% RSLogix 500 project Mixing_Room_1980_Kettle_original_backup_Aug_20_2021.RSS, saved by version 11.00.00.00 %
PROJECT "UNTITLED"    % processor: MicroLogix 1200 %

PROGRAM FILES
  LAD 2   55 rungs

DATA FILES
  O0 OUTPUT  8 elements
  I1 INPUT  13 elements
  S2 STATUS  66 elements
  B3 BINARY  5 elements
  T4 TIMER  5 elements
  C5 COUNTER  1 elements
  R6 CONTROL  1 elements
  N7 INTEGER  60 elements
  F8 FLOAT  141 elements
  PD9   1 elements

LADDER 2
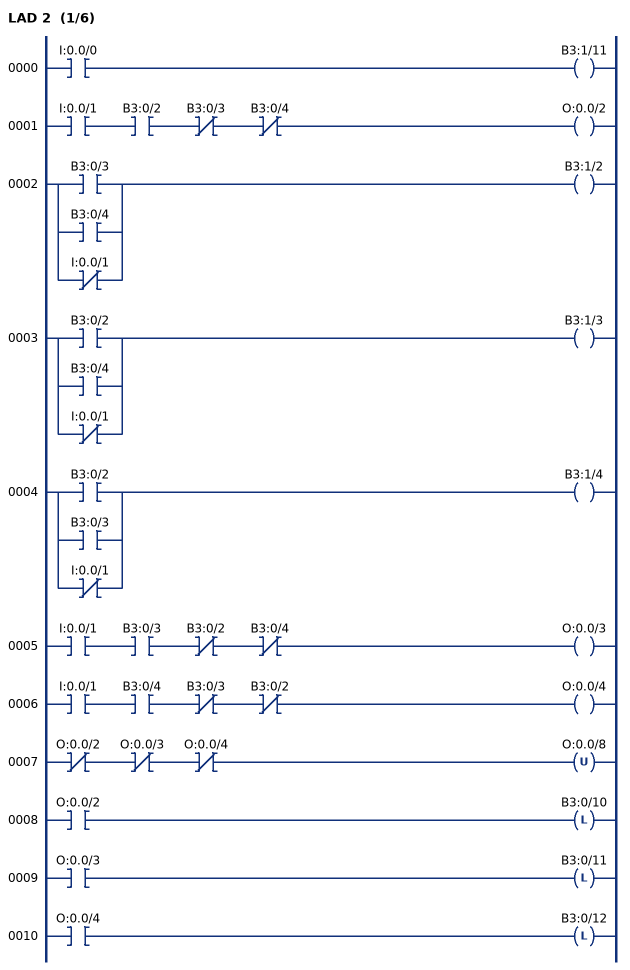
% Rung: 0 %
SOR XIC I:0.0/0 OTE B3:1/11 EOR
% Rung: 1 %
SOR XIC I:0.0/1 XIC B3:0/2 XIO B3:0/3 XIO B3:0/4 OTE O:0.0/2 EOR
% Rung: 2 %
SOR BST XIC B3:0/3 NXB BST XIC B3:0/4 NXB XIO I:0.0/1 BND BND OTE B3:1/2 EOR
% Rung: 3 %
SOR BST XIC B3:0/2 NXB BST XIC B3:0/4 NXB XIO I:0.0/1 BND BND OTE B3:1/3 EOR
% Rung: 4 %
SOR BST XIC B3:0/2 NXB BST XIC B3:0/3 NXB XIO I:0.0/1 BND BND OTE B3:1/4 EOR
% Rung: 5 %
SOR XIC I:0.0/1 XIC B3:0/3 XIO B3:0/2 XIO B3:0/4 OTE O:0.0/3 EOR
% Rung: 6 %
SOR XIC I:0.0/1 XIC B3:0/4 XIO B3:0/3 XIO B3:0/2 OTE O:0.0/4 EOR
% Rung: 7 %
SOR XIO O:0.0/2 XIO O:0.0/3 XIO O:0.0/4 OTU O:0.0/8 EOR
% Rung: 8 %
SOR XIC O:0.0/2 OTL B3:0/10 EOR
% Rung: 9 %
SOR XIC O:0.0/3 OTL B3:0/11 EOR
% Rung: 10 %
SOR XIC O:0.0/4 OTL B3:0/12 EOR

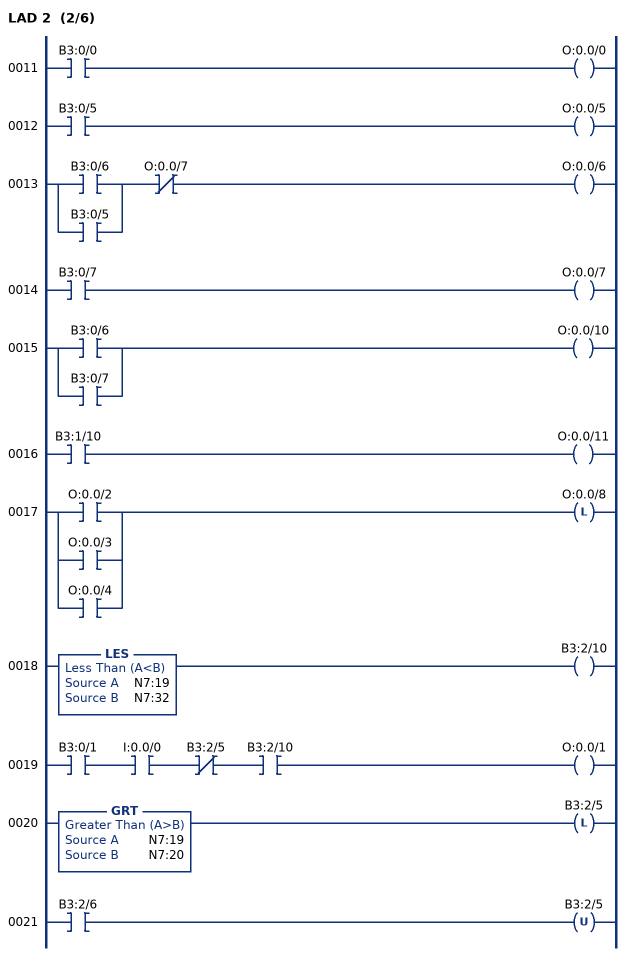
% Rung: 11 %
SOR XIC B3:0/0 OTE O:0.0/0 EOR
% Rung: 12 %
SOR XIC B3:0/5 OTE O:0.0/5 EOR
% Rung: 13 %
SOR BST XIC B3:0/6 NXB XIC B3:0/5 BND XIO O:0.0/7 OTE O:0.0/6 EOR
% Rung: 14 %
SOR XIC B3:0/7 OTE O:0.0/7 EOR
% Rung: 15 %
SOR BST XIC B3:0/6 NXB XIC B3:0/7 BND OTE O:0.0/10 EOR
% Rung: 16 %
SOR XIC B3:1/10 OTE O:0.0/11 EOR
% Rung: 17 %
SOR BST XIC O:0.0/2 NXB BST XIC O:0.0/3 NXB XIC O:0.0/4 BND BND OTL O:0.0/8 EOR
% Rung: 18 %
SOR LES N7:19 N7:32 OTE B3:2/10 EOR
% Rung: 19 %
SOR XIC B3:0/1 XIC I:0.0/0 XIO B3:2/5 XIC B3:2/10 OTE O:0.0/1 EOR
% Rung: 20 %
SOR GRT N7:19 N7:20 OTL B3:2/5 EOR
% Rung: 21 %
SOR XIC B3:2/6 OTU B3:2/5 EOR

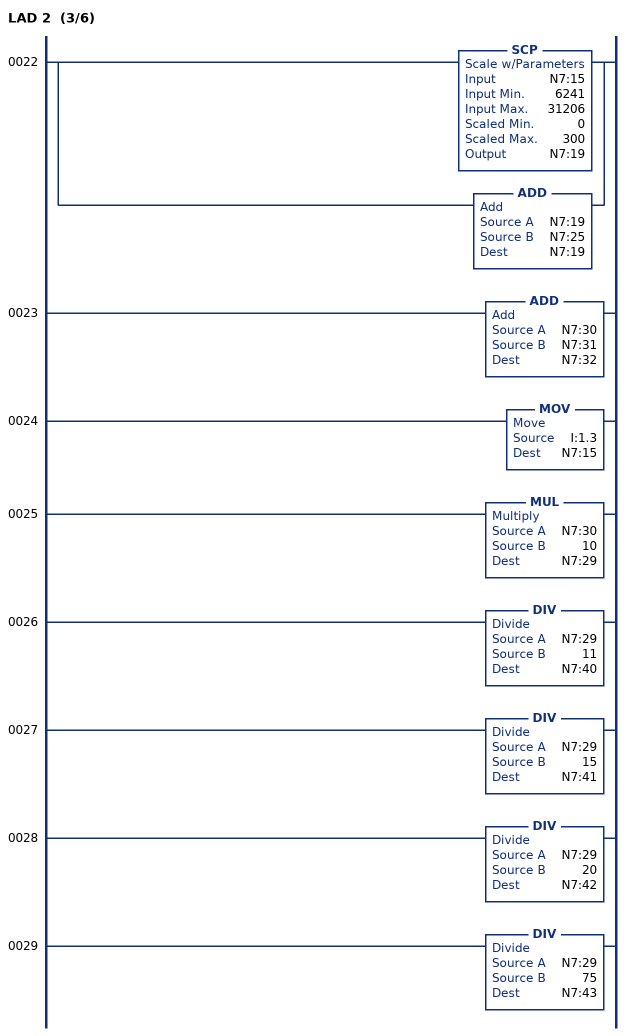
% Rung: 22 %
SOR BST SCP N7:15 6241 31206 0 300 N7:19 NXB ADD N7:19 N7:25 N7:19 BND EOR
% Rung: 23 %
SOR ADD N7:30 N7:31 N7:32 EOR
% Rung: 24 %
SOR MOV I:1.3 N7:15 EOR
% Rung: 25 %
SOR MUL N7:30 10 N7:29 EOR
% Rung: 26 %
SOR DIV N7:29 11 N7:40 EOR
% Rung: 27 %
SOR DIV N7:29 15 N7:41 EOR
% Rung: 28 %
SOR DIV N7:29 20 N7:42 EOR
% Rung: 29 %
SOR DIV N7:29 75 N7:43 EOR

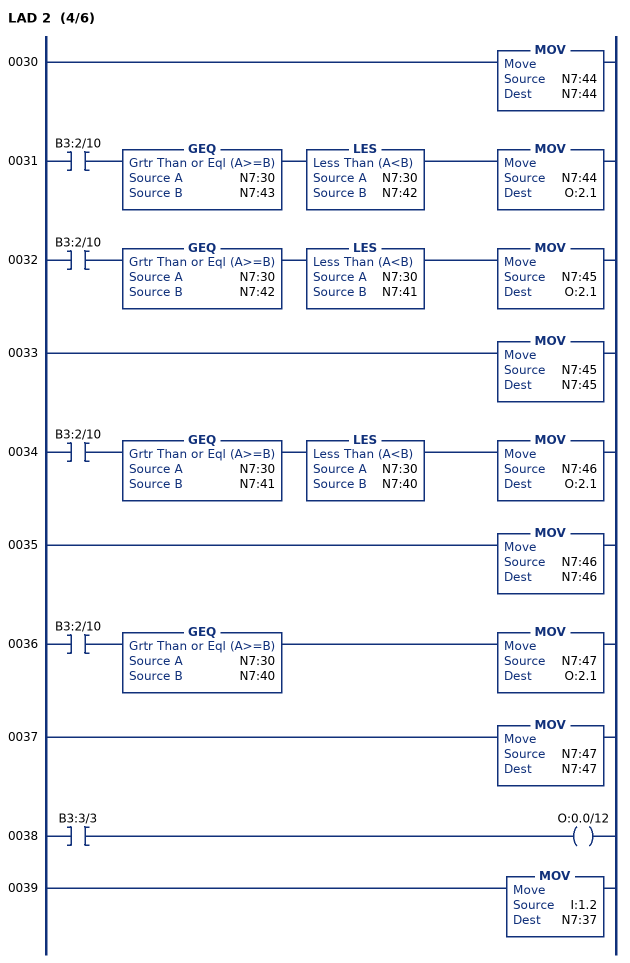
% Rung: 30 %
SOR MOV N7:44 N7:44 EOR
% Rung: 31 %
SOR XIC B3:2/10 GEQ N7:30 N7:43 LES N7:30 N7:42 MOV N7:44 O:2.1 EOR
% Rung: 32 %
SOR XIC B3:2/10 GEQ N7:30 N7:42 LES N7:30 N7:41 MOV N7:45 O:2.1 EOR
% Rung: 33 %
SOR MOV N7:45 N7:45 EOR
% Rung: 34 %
SOR XIC B3:2/10 GEQ N7:30 N7:41 LES N7:30 N7:40 MOV N7:46 O:2.1 EOR
% Rung: 35 %
SOR MOV N7:46 N7:46 EOR
% Rung: 36 %
SOR XIC B3:2/10 GEQ N7:30 N7:40 MOV N7:47 O:2.1 EOR
% Rung: 37 %
SOR MOV N7:47 N7:47 EOR
% Rung: 38 %
SOR XIC B3:3/3 OTE O:0.0/12 EOR
% Rung: 39 %
SOR MOV I:1.2 N7:37 EOR

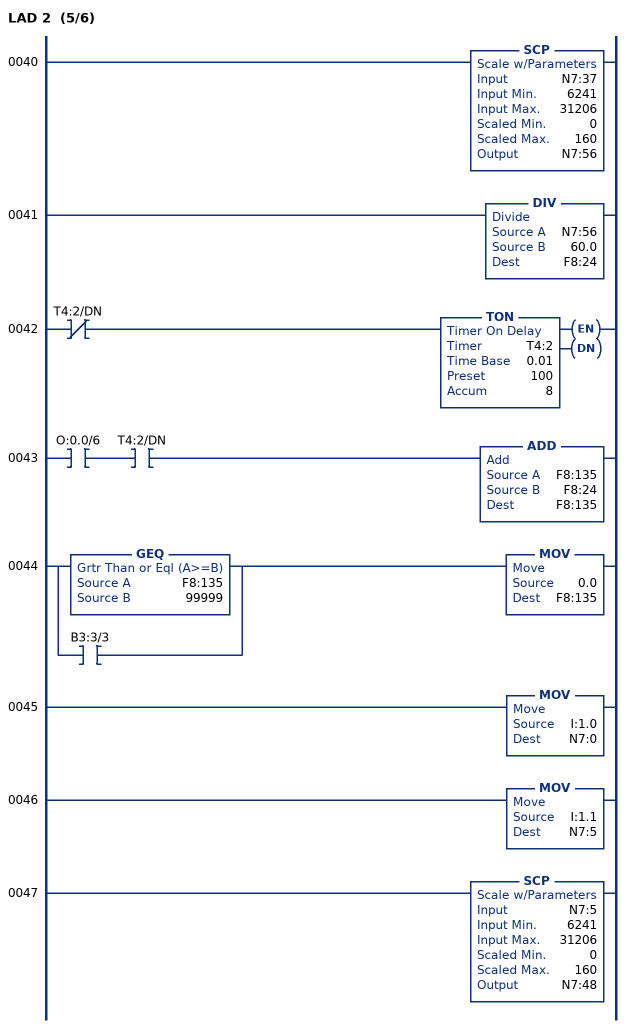
% Rung: 40 %
SOR SCP N7:37 6241 31206 0 160 N7:56 EOR
% Rung: 41 %
SOR DIV N7:56 60.0 F8:24 EOR
% Rung: 42 %
SOR XIO T4:2/DN TON T4:2 0.01 100 8 EOR
% Rung: 43 %
SOR XIC O:0.0/6 XIC T4:2/DN ADD F8:135 F8:24 F8:135 EOR
% Rung: 44 %
SOR BST GEQ F8:135 99999 NXB XIC B3:3/3 BND MOV 0.0 F8:135 EOR
% Rung: 45 %
SOR MOV I:1.0 N7:0 EOR
% Rung: 46 %
SOR MOV I:1.1 N7:5 EOR
% Rung: 47 %
SOR SCP N7:5 6241 31206 0 160 N7:48 EOR

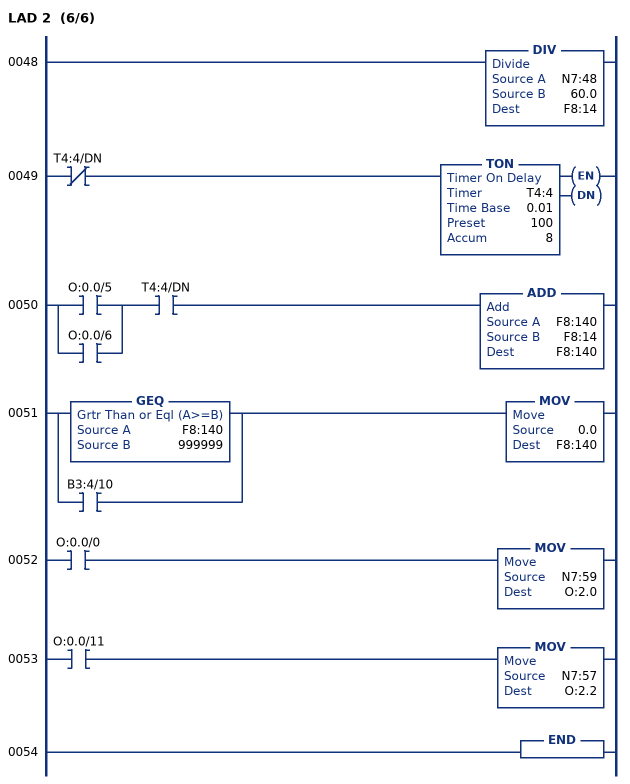
% Rung: 48 %
SOR DIV N7:48 60.0 F8:14 EOR
% Rung: 49 %
SOR XIO T4:4/DN TON T4:4 0.01 100 8 EOR
% Rung: 50 %
SOR BST XIC O:0.0/5 NXB XIC O:0.0/6 BND XIC T4:4/DN ADD F8:140 F8:14 F8:140 EOR
% Rung: 51 %
SOR BST GEQ F8:140 999999 NXB XIC B3:4/10 BND MOV 0.0 F8:140 EOR
% Rung: 52 %
SOR XIC O:0.0/0 MOV N7:59 O:2.0 EOR
% Rung: 53 %
SOR XIC O:0.0/11 MOV N7:57 O:2.2 EOR
% Rung: 54 %
SOR END EOR

DATA TABLE (non-zero values as saved)
DATA B3
% B3:0 % 0X1C00 0X0800 0X0400 0X0000 0X0000
DATA T4
% .PRE .ACC %
% T4:1 % 15 0
% T4:2 % 100 8
% T4:4 % 100 8
DATA N7
% N7:0 % 12047 135 100 1 0 6231 1 1 1 -52
% N7:10 % 12826 1 1 1 313 12174 135 1 1 71
% N7:20 % 230 0 0 0 0 0 0 0 0 1900
% N7:30 % 190 1 191 0 0 0 0 110 0 0
% N7:40 % 173 127 95 25 16510 25001 30001 31001 0 0
% N7:50 % 0 0 0 0 0 0 -39 20471 0 19722
DATA F8
% F8:20 % 0 0 0 0 -0.65
% F8:135 % -5661.661 0 0 0 0
% F8:140 % 328.4156
